{attribute 'linkalways'} 
{attribute 'no_explicit_call' := 'This FB is a CLASS and must be accessed using methods or properties'}
{attribute 'enable_dynamic_creation'}
FUNCTION_BLOCK _ULINT EXTENDS NumericDatatypeBase IMPLEMENTS I_ULINT
VAR
	localData : ULINT;
	activeData : REFERENCE TO ULINT REF= localData;
END_VAR

PROPERTY PUBLIC Address : PVOID
GET
Address := ADR(activeData);
END_GET
END_PROPERTY

METHOD PUBLIC ClearReference
VAR_INPUT
END_VAR
activeData REF= localData;
END_METHOD

METHOD PUBLIC Clone : I_Datatype
VAR
    pClone : POINTER TO _ULINT;
END_VAR
pClone := __NEW(_ULINT(InitialValue := Value));
Clone := pClone^;
END_METHOD

METHOD FB_init : BOOL
VAR_INPUT
	bInitRetains : BOOL; // if TRUE, the retain variables are initialized (warm start / cold start)
	bInCopyCode : BOOL;  // if TRUE, the instance afterwards gets moved into the copy code (online change)
	InitialValue : ULINT;
END_VAR
localData := InitialValue;
END_METHOD

PROPERTY PUBLIC IsEven : BOOL
GET
IsEven := (Value mod 2) = 0;
END_GET
END_PROPERTY

PROPERTY PUBLIC IsFloat : BOOL
GET
IsFloat := FALSE;
END_GET
END_PROPERTY

PROPERTY PUBLIC IsSigned : BOOL
GET
IsSigned := FALSE;
END_GET
END_PROPERTY

METHOD PUBLIC MakeReferenceTo
VAR_INPUT
	ReferenceTarget : REFERENCE TO ULINT;
END_VAR
activeData REF= ReferenceTarget;
END_METHOD

PROPERTY PUBLIC MaxValue : ULINT
GET
MaxValue :=  DatatypeLimits.ULINT_MAX_VALUE;
END_GET
END_PROPERTY

PROPERTY PUBLIC MinValue : ULINT
GET
MinValue := DatatypeLimits.ULINT_MIN_VALUE;
END_GET
END_PROPERTY

METHOD PROTECTED SerializeMaxValue
VAR_INPUT
	Serializer : I_Serializer;
END_VAR
Serializer.AddUlint(MaxValue);
END_METHOD

METHOD PROTECTED SerializeMinValue
VAR_INPUT
	Serializer : I_Serializer;
END_VAR
Serializer.AddUlint(MinValue);
END_METHOD

METHOD PUBLIC SerializeWith
VAR_INPUT
	Serializer : I_Serializer;
END_VAR
Serializer.AddUlint(activeData);
END_METHOD

PROPERTY PUBLIC Size : UDINT
GET
Size := SIZEOF(activeData);
END_GET
END_PROPERTY

METHOD PUBLIC TryConvertTo : BOOL
VAR_INPUT
	Destination : ANY;
END_VAR
TryConvertTo := TryConvert_ULINT_TO_Destination(activeData, Destination);
END_METHOD

METHOD PUBLIC TryConvertTo_ : BOOL
VAR_INPUT
	Destination : I_Datatype;
END_VAR
VAR
	resultofBitConversion : BOOL;
	destinationAs_BIT : I_BIT;
	destinationAs_BOOL : I_BOOL;
	destinationAs_BYTE : I_BYTE;
	destinationAs_DINT : I_DINT;
	destinationAs_DT : I_DT;
	destinationAs_DWORD : I_DWORD;
	destinationAs_INT : I_INT;
	destinationAs_LINT : I_LINT;
	destinationAs_LREAL : I_LREAL;
	destinationAs_LWORD : I_LWORD;
	destinationAs_REAL : I_REAL;
	destinationAs_SINT : I_SINT;
	destinationAs_STRING : I_STRING;
	destinationAs_TOD : I_TOD;
	destinationAs_UDINT : I_UDINT;
	destinationAs_UINT : I_UINT;
	destinationAs_ULINT : I_ULINT;
	destinationAs_USINT : I_USINT;
	destinationAs_WORD : I_WORD;
END_VAR
IF destination.TryResolveAs_BIT(destinationAs_BIT) AND_THEN TryConvert_ULINT_TO_BOOL(activeData, resultofBitConversion) THEN
	destinationAs_BIT.Value := resultOfBitConversion;
	TryConvertTo_ := TRUE;
	RETURN;
END_IF

IF destination.TryResolveAs_BOOL(destinationAs_BOOL) THEN
	TryConvertTo_ := TryConvert_ULINT_TO_BOOL(activeData, destinationAs_BOOL.Value);
	RETURN;
END_IF
		
IF destination.TryResolveAs_BYTE(destinationAs_BYTE) THEN
	TryConvertTo_ := TryConvert_ULINT_TO_BYTE(activeData, destinationAs_BYTE.Value);
	RETURN;
END_IF

IF destination.TryResolveAs_DINT(destinationAs_DINT) THEN
	TryConvertTo_ := TryConvert_ULINT_TO_DINT(activeData, destinationAs_DINT.Value);
	RETURN;
END_IF

IF destination.TryResolveAs_DT(destinationAs_DT) THEN
	TryConvertTo_ := TryConvert_ULINT_TO_DT(activeData, destinationAs_DT.Value);
	RETURN;
END_IF

IF destination.TryResolveAs_DWORD(destinationAs_DWORD) THEN
	TryConvertTo_ := TryConvert_ULINT_TO_DWORD(activeData, destinationAs_DWORD.Value);
	RETURN;
END_IF

IF destination.TryResolveAs_INT(destinationAs_INT) THEN
	TryConvertTo_ := TryConvert_ULINT_TO_INT(activeData, destinationAs_INT.Value);
	RETURN;
END_IF

IF destination.TryResolveAs_LINT(destinationAs_LINT) THEN
	TryConvertTo_ := TryConvert_ULINT_TO_LINT(activeData, destinationAs_LINT.Value);
	RETURN;
END_IF

IF destination.TryResolveAs_LREAL(destinationAs_LREAL) THEN
	TryConvertTo_ := TryConvert_ULINT_TO_LREAL(activeData, destinationAs_LREAL.Value);
	RETURN;
END_IF

IF destination.TryResolveAs_LWORD(destinationAs_LWORD) THEN
	TryConvertTo_ := TryConvert_ULINT_TO_LWORD(activeData, destinationAs_LWORD.Value);
	RETURN;
END_IF

IF destination.TryResolveAs_REAL(destinationAs_REAL) THEN
	TryConvertTo_ := TryConvert_ULINT_TO_REAL(activeData, destinationAs_REAL.Value);
	RETURN;
END_IF

IF destination.TryResolveAs_SINT(destinationAs_SINT) THEN
	TryConvertTo_ := TryConvert_ULINT_TO_SINT(activeData, destinationAs_SINT.Value);
	RETURN;
END_IF

IF destination.TryResolveAs_STRING(destinationAs_STRING) THEN
	TryConvertTo_ := TryConvert_ULINT_TO_STRING(activeData, destinationAs_STRING.Value);
	RETURN;
END_IF

IF destination.TryResolveAs_TOD(destinationAs_TOD) THEN
	TryConvertTo_ := TryConvert_ULINT_TO_TOD(activeData, destinationAs_TOD.Value);
	RETURN;
END_IF

IF destination.TryResolveAs_UDINT(destinationAs_UDINT) THEN
	TryConvertTo_ := TryConvert_ULINT_TO_UDINT(activeData, destinationAs_UDINT.Value);
	RETURN;
END_IF

IF destination.TryResolveAs_UINT(destinationAs_UINT) THEN
	TryConvertTo_ := TryConvert_ULINT_TO_UINT(activeData, destinationAs_UINT.Value);
	RETURN;
END_IF

IF destination.TryResolveAs_ULINT(destinationAs_ULINT) THEN
	TryConvertTo_ := TryConvert_ULINT_TO_ULINT(activeData, destinationAs_ULINT.Value);
	RETURN;
END_IF

IF destination.TryResolveAs_USINT(destinationAs_USINT) THEN
	TryConvertTo_ := TryConvert_ULINT_TO_USINT(activeData, destinationAs_USINT.Value);
	RETURN;
END_IF

IF destination.TryResolveAs_WORD(destinationAs_WORD) THEN
	TryConvertTo_ := TryConvert_ULINT_TO_WORD(activeData, destinationAs_WORD.Value);
	RETURN;
END_IF
END_METHOD

METHOD TryDeserializeFrom : BOOL
VAR_INPUT
	Deserializer : I_Deserializer;
	Feedback : I_DeserializerFeedback;
END_VAR
TryDeserializeFrom := Deserializer.TryGetUlint(activeData, Feedback);
END_METHOD

METHOD TryMakeReferenceTo : BOOL
VAR_INPUT
	Target : I_Datatype;
END_VAR
VAR
	pTargetData : POINTER TO ULINT;
END_VAR
IF NOT IsEquivalentTo(Target) THEN
	RETURN;
END_IF

pTargetData := Target.Address;
activeData REF= pTargetData^;
TryMakeReferenceTo := TRUE;
END_METHOD

METHOD PUBLIC TryResolveAs_ULINT : BOOL
VAR_INPUT
	Destination : REFERENCE TO I_ULINT;
END_VAR
Destination := THIS^;
TryResolveAs_ULINT := TRUE;
END_METHOD

PROPERTY PUBLIC TypeName : T_MAXSTRING
GET
TypeName := 'ULINT';
END_GET
END_PROPERTY

PROPERTY PUBLIC Value : REFERENCE TO ULINT
GET
Value REF= activeData;
END_GET
END_PROPERTY

END_FUNCTION_BLOCK

(* stored: Version 1.1.0.1, ProductVersion 3.1.4024.15
   POU _ULINT: Id {bde6120f-6364-4026-b44b-2fc58e406905}, SpecialFunc None
   Folder Constructor: Id {a72f9151-4509-46ce-a014-414877d198d4}
   Folder Protected: Id {435cb737-a039-4cff-8147-96d1f7bfc00f}
   Property Address: Id {82e246ac-c454-4c0d-803c-bc5bd0fbfb37}
   Get Get: Id {b048b36e-0738-4600-a8e4-722ca72aeb26}
   Method ClearReference: Id {41be9bb3-762e-4b07-a00c-1b91d469d5ec}
   Method Clone: Id {c51cdf13-1b01-4ad7-854d-70940ac8281d}
   Method FB_init: Id {513f7a59-3db1-4ce9-a741-3aea675fd306}
   Property IsEven: Id {b8c9b3d0-56a3-0114-0ed6-b2948bc39887}
   Get Get: Id {053892cc-6362-0628-1c02-4079d6b4cc8f}
   Property IsFloat: Id {fa2ffdb8-e5f6-47c5-b226-dce19e204ff6}
   Get Get: Id {259f0726-c668-4d66-973f-998347013f10}
   Property IsSigned: Id {36fc749e-eb6a-4c3f-b4a0-46b6cb0e9eef}
   Get Get: Id {fdda4534-5126-40e9-b63e-6b1e52e04ce0}
   Method MakeReferenceTo: Id {166cc47d-30de-46fb-9cb4-7e6d50154009}
   Property MaxValue: Id {e8951ca6-eb4d-4551-9eab-45fa00e85acc}
   Get Get: Id {c63b0f4c-c92b-4f86-a014-c2f166de1a3b}
   Property MinValue: Id {0ecb9636-31ec-4de8-8419-dd61e1781db9}
   Get Get: Id {ec8b3d9a-8ccd-4247-afb5-7ff5b16b7c8a}
   Method SerializeMaxValue: Id {95e46651-ff87-4a8c-8d42-2b7eeb850a42}
   Method SerializeMinValue: Id {3bbf25ba-79ad-45a3-a4fe-024e5a3f818d}
   Method SerializeWith: Id {af52ddc8-39c0-4982-a867-7d2707e5c981}
   Property Size: Id {c8005a4d-c7ea-458b-80de-07da5a24f0d6}
   Get Get: Id {861ccdff-d8ad-4f6a-9bfc-8f22117bf83e}
   Method TryConvertTo: Id {d0c890bb-27b3-0079-0b28-04a58e214385}
   Method TryConvertTo_: Id {84cf51c5-e59e-01ac-10df-eb8f469fdf79}
   Method TryDeserializeFrom: Id {c16a4453-72b9-4acf-a58a-b1d5b7e37d83}
   Method TryMakeReferenceTo: Id {fef61275-13e2-4cbb-b370-403774d8bbca}
   Method TryResolveAs_ULINT: Id {6792d707-5bb9-0683-29cb-8e0290f2548a}
   Property TypeName: Id {fdc4282b-f205-42f3-8e27-650dc9a0c240}
   Get Get: Id {e5ac2442-aefc-4db6-87ce-fdc6b59e7d21}
   Property Value: Id {d8357b2b-85f4-473a-935d-9f2911300336}
   Get Get: Id {c3875205-357f-4f79-aa96-fa4036973510} *)
